{attribute 'qualified_only'}
VAR_GLOBAL
	/// Inputs
	bHomeSwitch 		AT %I* : BOOL;
	/// Outputs
	
END_VAR

(* stored: Version 1.1.0.1, ProductVersion 3.1.4024.12
   GVL IO: Id {ec8b3721-9de7-4a16-b80d-24d091a4ea63} *)
